Yaskawa INFORM job: GO-TO-PARK-POS-DEMO-PRG.JBI

/JOB
//NAME GO-TO-PARK-POS-DEMO-PRG
//POS
///NPOS 1,0,0,1,0,0
///TOOL 0
///POSTYPE PULSE
///PULSE
C00000=-107423,-36358,10351,68056,-126377,117727
///USER 10
///POSTYPE USER
///RECTAN
///RCONF 0,0,0,0,0,0,0,0,0,0,0,0,0,0,0,0,0,0,0,0,0,0,0,0
P00162=200.000,0.000,0.000,0.0000,0.0000,0.0000
//INST
///DATE 2018/10/05 07:50
///ATTR SC,RW
///GROUP1 RB1
NOP
DOUT OT#(22) OFF
'*****
SETE P0162 (1) -200000
IMOV P0162 V=250.0 UF#(10)
'*****
MOVJ C00000 VJ=25.00
'*****
SETREG MREG#(1) 11
END
